{attribute 'qualified_only'}
{attribute 'strict'}
TYPE E_Color :
(
	enum_member := 0
);
END_TYPE

(* stored: Version 1.1.0.1, ProductVersion 3.1.4024.12
   DUT E_Color: Id {e2c7da18-9138-4ef6-a531-74258d576d7d} *)
